FUNCTION_BLOCK FB_Encoder_Test EXTENDS FB_TestSuite
VAR	
	stConfig 			: ST_EncoderConfig;
END_VAR

TestCase_Encoder('Absolute 1', 0, 0, LREAL_TO_DINT(0*1E4), stConfig);
TestCase_Encoder('Absolute 2', 100, 100, LREAL_TO_DINT(100*1E4), stConfig);
TestCase_Encoder('Absolute 3', -100, -100, LREAL_TO_DINT(-100*1E4), stConfig);

stConfig.fInputFactor := -1;
TestCase_Encoder('Absolute with Factor 1', 0, 0, LREAL_TO_DINT(0*1E4), stConfig);
TestCase_Encoder('Absolute with Factor 2', 100, -100, LREAL_TO_DINT(-100*1E4), stConfig);
TestCase_Encoder('Absolute with Factor 3', -100, 100, LREAL_TO_DINT(100*1E4), stConfig);

stConfig.fInputFactor := 1;
stConfig.bInvertIncrementValue := TRUE;
TestCase_Encoder('Absolute with Invert 1', 0, 0, LREAL_TO_DINT(0*1E4), stConfig);
TestCase_Encoder('Absolute with Invert 2', 100, 100, LREAL_TO_DINT(-100*1E4), stConfig);
TestCase_Encoder('Absolute with Invert 3', -100, -100, LREAL_TO_DINT(100*1E4), stConfig);

stConfig.fModulo := 360;
stConfig.bInvertIncrementValue := FALSE;
TestCase_Encoder('Modulo 1', 0, 0, LREAL_TO_DINT(0*1E4), stConfig);
TestCase_Encoder('Modulo 2', 360, 0, LREAL_TO_DINT(0*1E4), stConfig);
TestCase_Encoder('Modulo 3', 350, 350, LREAL_TO_DINT(350*1E4), stConfig);
TestCase_Encoder('Modulo 4', -350, -350, LREAL_TO_DINT(-350*1E4), stConfig);
TestCase_Encoder('Modulo 5', -360, 0, LREAL_TO_DINT(0*1E4), stConfig);

stConfig.fModulo := 0;
stConfig.bInvertIncrementValue := FALSE;
stConfig.bIsIntegral := TRUE;
TestCase_Encoder('Integrate 1', 0, 0, 0, stConfig);
TestCase_Encoder('Integrate 2', 100, 1, LREAL_TO_DINT(1*1E4), stConfig);
TestCase_Encoder('Integrate 3', -100, -1, LREAL_TO_DINT(-1*1E4), stConfig);

METHOD TestCase_Encoder
VAR_INPUT
	sName 					: T_MaxString;
	fInput					: REAL;
	fExpected				: LREAL;
	nExpected				: DINT;
	stConfig				: ST_EncoderConfig;
END_VAR

VAR	
	fbEncoder 				: FB_Encoder;
	nCycleCount 			: INT;
	fActual					: LREAL;	
	nActual					: DINT;	
	bValid 					: BOOL;
	fTolerance 				: REAL := 1E-6;
END_VAR
TEST(sName);

fbEncoder.stConfig := stConfig;
fbEncoder.fInput := fInput;

(*	Call FB to test	*)
FOR nCycleCount := 0 TO 9 DO
   fbEncoder();
END_FOR

(*	Evaluation of results	*)
nActual := fbEncoder.nPosition;
fActual := fbEncoder.fPosition;

AssertEquals(Expected := nExpected,
             Actual := nActual,
             Message := 'nPosition is not correct');

bValid := ABS(fExpected - fActual) < fTolerance;			 
	
AssertTrue(bValid, 'fPosition is not correct');

TEST_FINISHED();
END_METHOD

END_FUNCTION_BLOCK

(* stored: Version 1.1.0.1, ProductVersion 3.1.4024.12
   POU FB_Encoder_Test: Id {2e2b1666-3023-0dca-3449-a99196318ada}, SpecialFunc None
   Method TestCase_Encoder: Id {dc10b32a-3ed5-0a79-0d3c-95258e3cf3ee} *)
